FUNCTION_BLOCK E_SPLIT3
  (* Version 1.0, 2005-06-24, Goran Cengic, Chalmers *)
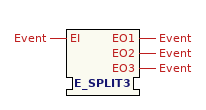
  EVENT_INPUT
    EI;
  END_EVENT
  EVENT_OUTPUT
    EO1;
    EO2;
    EO3;
  END_EVENT
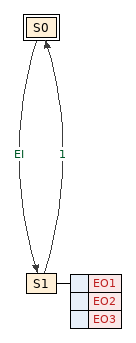
  EC_STATES
    S0;
    S1 : -> EO1, -> EO2, -> EO3;
  END_STATES
  EC_TRANSITIONS
    S0 TO S1 := EI;
    S1 TO S0 := 1;
  END_TRANSITIONS
END_FUNCTION_BLOCK
